FUNCTION_BLOCK TcoPlbPaletizator_Positions EXTENDS TcoDrivesBeckhoff.TcoSingleAxisPositionsRootContainer
VAR_INPUT
END_VAR
VAR_OUTPUT
END_VAR
VAR

	
	{attribute addProperty Name "<#Pracovna pozicia#>"}
	WorkPosition : TcoDrivesBeckhoff.TcoMultiAxisMoveParam;
	{attribute addProperty Name "<#Naberacia pozicia Buffer1#>"}
	LoadFromBuffer1Postion : TcoDrivesBeckhoff.TcoMultiAxisMoveParam;
	{attribute addProperty Name "<#Naberacia pozicia Buffer2#>"}
	LoadFromBuffer2Postion : TcoDrivesBeckhoff.TcoMultiAxisMoveParam;
	{attribute addProperty Name "<#Naberacia pozicia Buffer3#>"}
	LoadFromBuffer3Postion : TcoDrivesBeckhoff.TcoMultiAxisMoveParam;
	{attribute addProperty Name "<#Naberacia pozicia Buffer4#>"}
	LoadFromBuffer4Postion : TcoDrivesBeckhoff.TcoMultiAxisMoveParam;
	{attribute addProperty Name "<#Vykladacia pozicia pre prazdne blistre 1#>"}
	UnloadEmpty1Postion : TcoDrivesBeckhoff.TcoMultiAxisMoveParam;
	{attribute addProperty Name "<#Vykladacia pozicia pre prazdne blistre 2#>"}
	UnloadEmpty2Postion : TcoDrivesBeckhoff.TcoMultiAxisMoveParam;

END_VAR

PROPERTY PUBLIC LoadFromBuffer1Pos : reference to TcoDrivesBeckhoff.TcoMultiAxisMoveParam;
GET
LoadFromBuffer1Pos ref=LoadFromBuffer1Postion;
END_GET
END_PROPERTY

PROPERTY PUBLIC LoadFromBuffer2Pos : reference to TcoDrivesBeckhoff.TcoMultiAxisMoveParam;
GET
LoadFromBuffer2Pos ref=LoadFromBuffer2Postion;
END_GET
END_PROPERTY

PROPERTY PUBLIC LoadFromBuffer3Pos : reference to TcoDrivesBeckhoff.TcoMultiAxisMoveParam;
GET
LoadFromBuffer3Pos ref=LoadFromBuffer3Postion;
END_GET
END_PROPERTY

PROPERTY PUBLIC LoadFromBuffer4Pos : reference to TcoDrivesBeckhoff.TcoMultiAxisMoveParam;
GET
LoadFromBuffer4Pos REF=LoadFromBuffer4Postion;
END_GET
END_PROPERTY

PROPERTY PUBLIC UnloadEmpty1Pos : reference to TcoDrivesBeckhoff.TcoMultiAxisMoveParam;
GET
UnloadEmpty1Pos REF=UnloadEmpty1Postion;
END_GET
END_PROPERTY

PROPERTY PUBLIC UnloadEmpty2Pos : reference to TcoDrivesBeckhoff.TcoMultiAxisMoveParam;
GET
UnloadEmpty2Pos REF=UnloadEmpty2Postion;
END_GET
END_PROPERTY

PROPERTY PUBLIC WorkPos : reference to TcoDrivesBeckhoff.TcoMultiAxisMoveParam;
GET
WorkPos ref= WorkPosition;
END_GET
END_PROPERTY

END_FUNCTION_BLOCK

(* stored: Version 1.1.0.1
   POU TcoPlbPaletizator_Positions: Id {c9f46cce-6c18-4669-ae24-84f55103b084}, SpecialFunc None
   Property LoadFromBuffer1Pos: Id {526cb63e-afa2-41b7-883d-49902dde54fe}
   Get Get: Id {41e21bbf-30f2-40ce-841c-e8c11a33ff29}
   Property LoadFromBuffer2Pos: Id {0702a3a7-c53c-4dfb-ae4f-02f5ac01e40c}
   Get Get: Id {de5dab8f-bc2d-4315-9836-112e46e36725}
   Property LoadFromBuffer3Pos: Id {71757d59-ff6b-41d9-ad40-35473985e7c7}
   Get Get: Id {2a723db0-a444-498d-a71e-ca7b0aed3145}
   Property LoadFromBuffer4Pos: Id {12cbbb34-1671-4fa4-81f0-bd41cf1f8d50}
   Get Get: Id {b1faea9f-29c2-47e8-b1a2-18f812686bec}
   Property UnloadEmpty1Pos: Id {cd844036-7951-42ac-a2b6-3ae839952bbf}
   Get Get: Id {3d346716-383e-49ac-860f-7636816f37c9}
   Property UnloadEmpty2Pos: Id {e0575526-80b9-40b5-a2a3-1ecb43c5b0a0}
   Get Get: Id {5991fb66-ab5d-470b-bab9-b6a4fbbba03b}
   Property WorkPos: Id {4a5ede3e-3e1f-4373-80ed-660253e25041}
   Get Get: Id {173303b9-a3e7-4a0f-b1c6-49e2108e4bcf} *)
